DATA_BLOCK "dbArchiveGroup"
{ S7_Optimized_Access := 'TRUE' }
VERSION : 0.8
NON_RETAIN
"fbArchiveGroup"

BEGIN

END_DATA_BLOCK

